PROGRAM EM04_Placing3
VAR
	
	//Backbone
	FB_StateMachine_Placing3		: FB_StateManager;
	bFl_RunningMachinePlacing3		: BOOL;
	bFl_SeqReset					: BOOL;
	bFl_Manual						: BOOL;
	CheckStatusPlacing3				: checkstatus;
	AlarmEventHistory				: ARRAY[1..20] OF Alarm_Event_History;
	Placing3_Management				: FB_Placing;
	bFl_Flushing					: BOOL;
	PalletID_Placing3				: PalletID_Name;
	Placing3_ID						: STRING;
	bFl_PalletJammed				: BOOL;
	
	//Motor
	Motor_PalletPlacing3			: MotorManagement;
	bFl_MotorPlacing3				: BOOL;
	Motor_Placing3_Error			: BOOL;
	Motor_Placing3_ErrorID			: UINT;
	bFl_MotorPlacing3_Fwd			: BOOL;
	bFl_MotorPlacing3_Rev			: BOOL;
	bFL_Safety						: BOOL;
	AlarmEventActive				: ARRAY[1..20] OF Alarm_Event_Active;
	CheckAcc						: TON;
END_VAR
VAR // added by the converter: edge detectors and wires of the graphical bodies
    _w1 : BOOL;
END_VAR

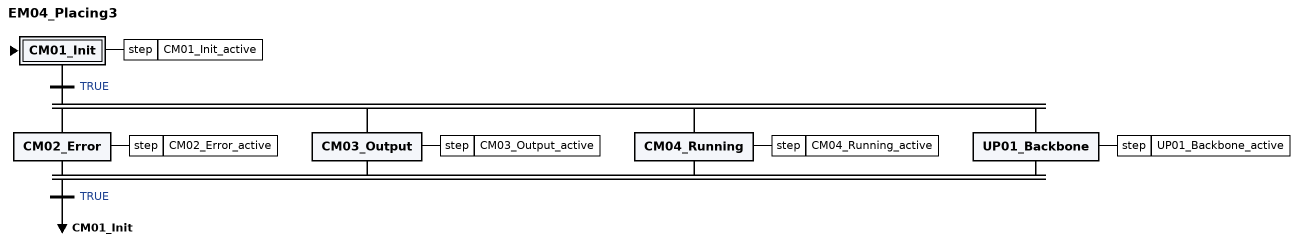
INITIAL_STEP CM01_Init:
    CM01_Init_active(N);  // step action
END_STEP
TRANSITION FROM CM01_Init TO (CM02_Error, CM03_Output, CM04_Running, UP01_Backbone)
    := TRUE;
END_TRANSITION
STEP CM02_Error:
    CM02_Error_active(N);  // step action
END_STEP
STEP CM03_Output:
    CM03_Output_active(N);  // step action
END_STEP
STEP CM04_Running:
    CM04_Running_active(N);  // step action
END_STEP
STEP UP01_Backbone:
    UP01_Backbone_active(N);  // step action
END_STEP
TRANSITION FROM (CM02_Error, CM03_Output, CM04_Running, UP01_Backbone) TO CM01_Init
    := TRUE;
END_TRANSITION

ACTION CM01_Init_active:
Data_GVL.bFL_StartPlacing3			:= Status_GVL.bFl_RunButton_Robotic OR HMI_GVL.bStartButtonPlacing3;
Data_GVL.bFL_StopPlacing3			:= NOT Status_GVL.bFl_StopButton_Robotic OR HMI_GVL.bStopButtonPlacing3;
Data_GVL.bFL_ResetPlacing3			:= Status_GVL.bFl_ResetButton_Robotic OR HMI_GVL.bResetButtonPlacing3;
Data_GVL.bFL_AckPlacing3			:= Status_GVL.bFl_Acknowledge_Robotic OR HMI_GVL.bAcknowledgeButtonPlacing3;
Data_GVL.bFL_AutoManuaModePlacing3 	:= Status_GVL.bFl_Manual_Robotic OR HMI_GVL.bTestModeEnablePlacing3;
bFl_RunningMachinePlacing3			:= Data_GVL.stStateMachinePlacing3.Running;
bFl_Manual							:= Data_GVL.stStateMachinePlacing3.ManualMode;
bFl_SeqReset						:= NOT Status_GVL.bFl_EStop_Robotic;
bFL_Safety							:= Status_GVL.bFl_EStop_Robotic AND Status_GVL.bSafety_DoorRobotic;


(*=================Convert Timer============================*)
Data_GVL.Tmr_Placing3	:= ConvertMilliSecTimeData(HMI_GVL.Tmr_Placing3);


(*=================Data OEE============================*)
Data_GVL.dt_Production[3].Data1			:= HMI_GVL.arCountTotal[3];
Data_GVL.dt_Production[3].Data2			:= HMI_GVL.arPalletTotal[3];
Data_GVL.dt_Production[3].Data3			:= HMI_GVL.arPalletIncomplete[3];
Data_GVL.dt_Production[3].ProductCode	:= Status_GVL.RecipeLine[3].ProductName;
END_ACTION

ACTION CM02_Error_active:
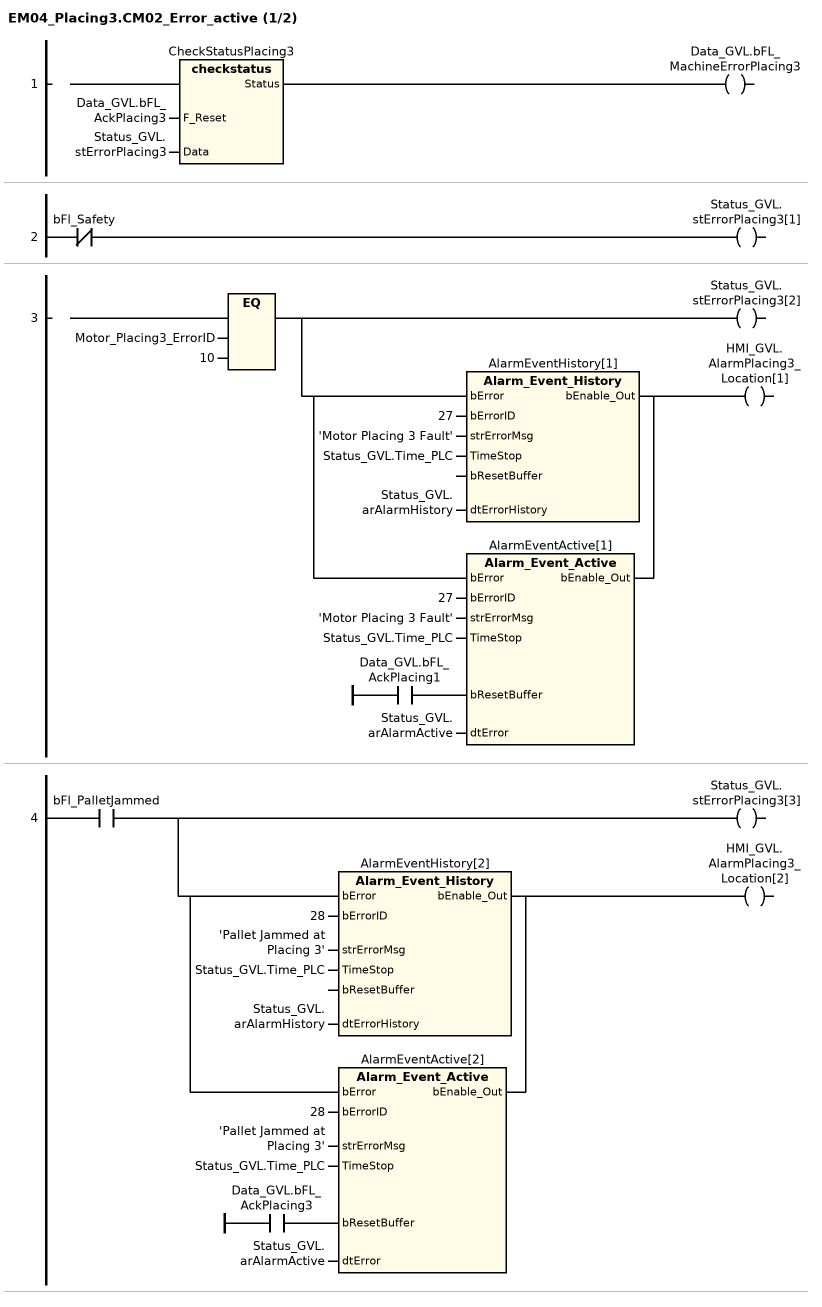
// NETWORK 1
CheckStatusPlacing3(F_Reset := Data_GVL.bFL_AckPlacing3, Data := Status_GVL.stErrorPlacing3); // checkstatus
Data_GVL.bFL_MachineErrorPlacing3 := CheckStatusPlacing3.Status;

// NETWORK 2
Status_GVL.stErrorPlacing3[1] := NOT bFl_Safety;

// NETWORK 3
_w1 := Motor_Placing3_ErrorID = 10;
Status_GVL.stErrorPlacing3[2] := _w1;
AlarmEventHistory[1](
    bError := _w1,
    bErrorID := 27,
    strErrorMsg := 'Motor Placing 3 Fault',
    TimeStop := Status_GVL.Time_PLC,
    dtErrorHistory := Status_GVL.arAlarmHistory); // Alarm_Event_History
AlarmEventActive[1](
    bError := _w1,
    bErrorID := 27,
    strErrorMsg := 'Motor Placing 3 Fault',
    TimeStop := Status_GVL.Time_PLC,
    bResetBuffer := Data_GVL.bFL_AckPlacing1,
    dtError := Status_GVL.arAlarmActive); // Alarm_Event_Active
HMI_GVL.AlarmPlacing3_Location[1] := AlarmEventHistory[1].bEnable_Out OR AlarmEventActive[1].bEnable_Out;

// NETWORK 4
Status_GVL.stErrorPlacing3[3] := bFl_PalletJammed;
AlarmEventHistory[2](
    bError := bFl_PalletJammed,
    bErrorID := 28,
    strErrorMsg := 'Pallet Jammed at Placing 3',
    TimeStop := Status_GVL.Time_PLC,
    dtErrorHistory := Status_GVL.arAlarmHistory); // Alarm_Event_History
AlarmEventActive[2](
    bError := bFl_PalletJammed,
    bErrorID := 28,
    strErrorMsg := 'Pallet Jammed at Placing 3',
    TimeStop := Status_GVL.Time_PLC,
    bResetBuffer := Data_GVL.bFL_AckPlacing3,
    dtError := Status_GVL.arAlarmActive); // Alarm_Event_Active
HMI_GVL.AlarmPlacing3_Location[2] := AlarmEventHistory[2].bEnable_Out OR AlarmEventActive[2].bEnable_Out;

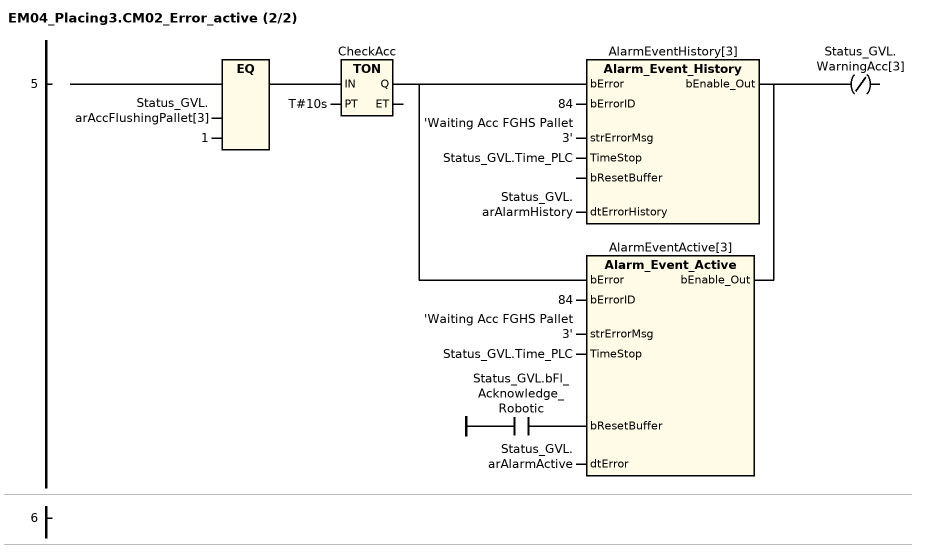
// NETWORK 5
CheckAcc(IN := Status_GVL.arAccFlushingPallet[3] = 1, PT := T#10s); // TON
AlarmEventHistory[3](
    bError := CheckAcc.Q,
    bErrorID := 84,
    strErrorMsg := 'Waiting Acc FGHS Pallet 3',
    TimeStop := Status_GVL.Time_PLC,
    dtErrorHistory := Status_GVL.arAlarmHistory); // Alarm_Event_History
AlarmEventActive[3](
    bError := CheckAcc.Q,
    bErrorID := 84,
    strErrorMsg := 'Waiting Acc FGHS Pallet 3',
    TimeStop := Status_GVL.Time_PLC,
    bResetBuffer := Status_GVL.bFl_Acknowledge_Robotic,
    dtError := Status_GVL.arAlarmActive); // Alarm_Event_Active
Status_GVL.WarningAcc[3] := NOT (AlarmEventHistory[3].bEnable_Out OR AlarmEventActive[3].bEnable_Out);

// NETWORK 6
END_ACTION

ACTION CM03_Output_active:
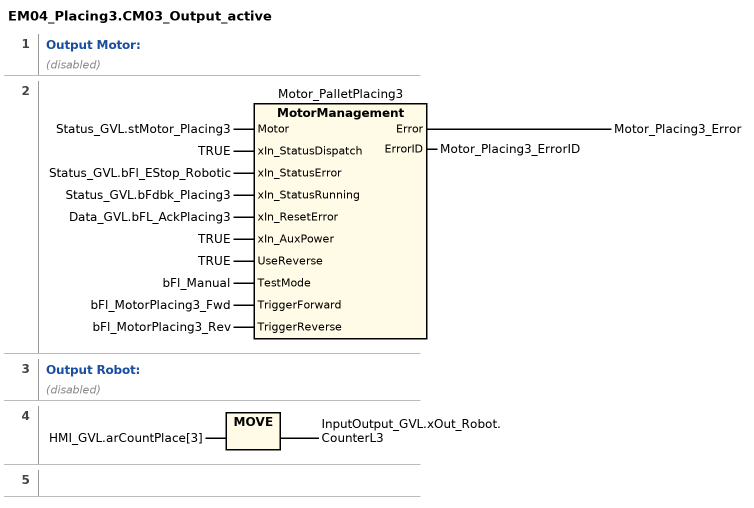
// NETWORK 1 (disabled)
// label: Output Motor

// NETWORK 2
Motor_PalletPlacing3(
    Motor := Status_GVL.stMotor_Placing3,
    xIn_StatusDispatch := TRUE,
    xIn_StatusError := Status_GVL.bFl_EStop_Robotic,
    xIn_StatusRunning := Status_GVL.bFdbk_Placing3,
    xIn_ResetError := Data_GVL.bFL_AckPlacing3,
    xIn_AuxPower := TRUE,
    UseReverse := TRUE,
    TestMode := bFl_Manual,
    TriggerForward := bFl_MotorPlacing3_Fwd,
    TriggerReverse := bFl_MotorPlacing3_Rev,
    ErrorID => Motor_Placing3_ErrorID); // MotorManagement
Motor_Placing3_Error := Motor_PalletPlacing3.Error;

// NETWORK 3 (disabled)
// label: Output Robot

// NETWORK 4
InputOutput_GVL.xOut_Robot.CounterL3 := HMI_GVL.arCountPlace[3];

// NETWORK 5
END_ACTION

ACTION CM04_Running_active:
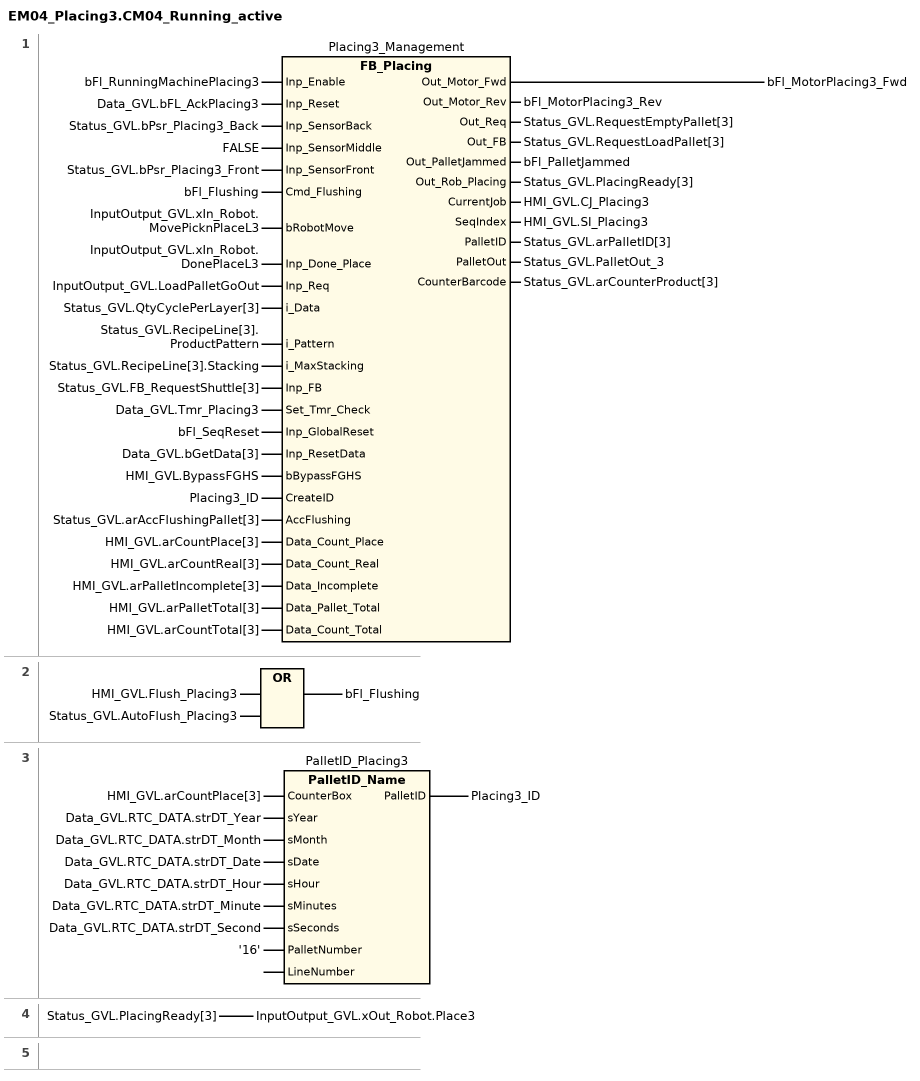
// NETWORK 1
Placing3_Management(
    Inp_Enable := bFl_RunningMachinePlacing3,
    Inp_Reset := Data_GVL.bFL_AckPlacing3,
    Inp_SensorBack := Status_GVL.bPsr_Placing3_Back,
    Inp_SensorMiddle := FALSE,
    Inp_SensorFront := Status_GVL.bPsr_Placing3_Front,
    Cmd_Flushing := bFl_Flushing,
    bRobotMove := InputOutput_GVL.xIn_Robot.MovePicknPlaceL3,
    Inp_Done_Place := InputOutput_GVL.xIn_Robot.DonePlaceL3,
    Inp_Req := InputOutput_GVL.LoadPalletGoOut,
    i_Data := Status_GVL.QtyCyclePerLayer[3],
    i_Pattern := Status_GVL.RecipeLine[3].ProductPattern,
    i_MaxStacking := Status_GVL.RecipeLine[3].Stacking,
    Inp_FB := Status_GVL.FB_RequestShuttle[3],
    Set_Tmr_Check := Data_GVL.Tmr_Placing3,
    Inp_GlobalReset := bFl_SeqReset,
    Inp_ResetData := Data_GVL.bGetData[3],
    bBypassFGHS := HMI_GVL.BypassFGHS,
    CreateID := Placing3_ID,
    AccFlushing := Status_GVL.arAccFlushingPallet[3],
    Data_Count_Place := HMI_GVL.arCountPlace[3],
    Data_Count_Real := HMI_GVL.arCountReal[3],
    Data_Incomplete := HMI_GVL.arPalletIncomplete[3],
    Data_Pallet_Total := HMI_GVL.arPalletTotal[3],
    Data_Count_Total := HMI_GVL.arCountTotal[3],
    Out_Motor_Rev => bFl_MotorPlacing3_Rev,
    Out_Req => Status_GVL.RequestEmptyPallet[3],
    Out_FB => Status_GVL.RequestLoadPallet[3],
    Out_PalletJammed => bFl_PalletJammed,
    Out_Rob_Placing => Status_GVL.PlacingReady[3],
    CurrentJob => HMI_GVL.CJ_Placing3,
    SeqIndex => HMI_GVL.SI_Placing3,
    PalletID => Status_GVL.arPalletID[3],
    PalletOut => Status_GVL.PalletOut_3,
    CounterBarcode => Status_GVL.arCounterProduct[3]); // FB_Placing
bFl_MotorPlacing3_Fwd := Placing3_Management.Out_Motor_Fwd;

// NETWORK 2
bFl_Flushing := HMI_GVL.Flush_Placing3 OR Status_GVL.AutoFlush_Placing3;

// NETWORK 3
PalletID_Placing3(
    CounterBox := HMI_GVL.arCountPlace[3],
    sYear := Data_GVL.RTC_DATA.strDT_Year,
    sMonth := Data_GVL.RTC_DATA.strDT_Month,
    sDate := Data_GVL.RTC_DATA.strDT_Date,
    sHour := Data_GVL.RTC_DATA.strDT_Hour,
    sMinutes := Data_GVL.RTC_DATA.strDT_Minute,
    sSeconds := Data_GVL.RTC_DATA.strDT_Second,
    PalletNumber := '16'); // PalletID_Name
Placing3_ID := PalletID_Placing3.PalletID;

// NETWORK 4
InputOutput_GVL.xOut_Robot.Place3 := Status_GVL.PlacingReady[3];

// NETWORK 5
END_ACTION

ACTION UP01_Backbone_active:
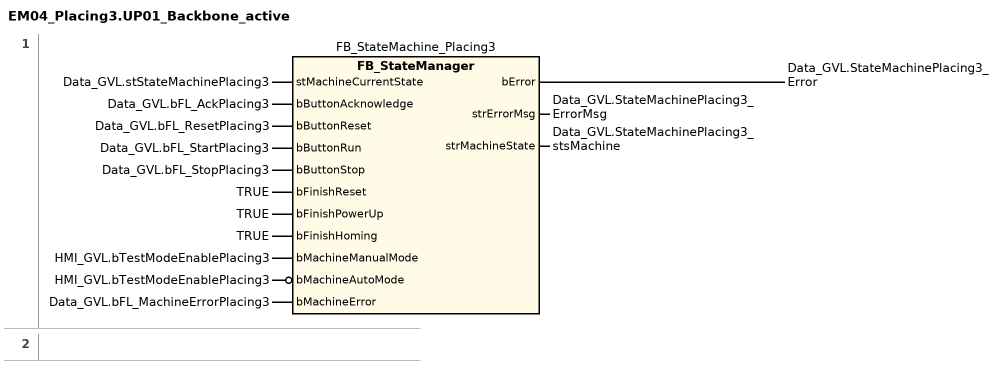
// NETWORK 1
FB_StateMachine_Placing3(
    stMachineCurrentState := Data_GVL.stStateMachinePlacing3,
    bButtonAcknowledge := Data_GVL.bFL_AckPlacing3,
    bButtonReset := Data_GVL.bFL_ResetPlacing3,
    bButtonRun := Data_GVL.bFL_StartPlacing3,
    bButtonStop := Data_GVL.bFL_StopPlacing3,
    bFinishReset := TRUE,
    bFinishPowerUp := TRUE,
    bFinishHoming := TRUE,
    bMachineManualMode := HMI_GVL.bTestModeEnablePlacing3,
    bMachineAutoMode := NOT HMI_GVL.bTestModeEnablePlacing3,
    bMachineError := Data_GVL.bFL_MachineErrorPlacing3,
    strErrorMsg => Data_GVL.StateMachinePlacing3_ErrorMsg,
    strMachineState => Data_GVL.StateMachinePlacing3_stsMachine); // FB_StateManager
Data_GVL.StateMachinePlacing3_Error := FB_StateMachine_Placing3.bError;

// NETWORK 2
END_ACTION

END_PROGRAM

(* stored: Version 1.1.0.1, ProductVersion 3.1.4024.12
   POU EM04_Placing3: Id {5a1718e7-4de1-4109-9549-66e6f35c5bc6}, SpecialFunc None
   Action CM01_Init_active: Id {9367e3fb-8aff-48d4-9106-0af4a50a15a8}
   Action CM02_Error_active: Id {37de86a5-d7b9-40eb-973a-96f62680b825}
   Action CM03_Output_active: Id {15dd54ee-f6dd-4197-8838-40785914e900}
   Action CM04_Running_active: Id {8c791cca-4183-48bf-a8de-d15976a3ebf6}
   Action UP01_Backbone_active: Id {d39eb8af-6fc4-43aa-812a-e8e3281c1228} *)
